# B&R Automation Studio project Laba_2
Automation Studio 4.2.5.388

## Configuration SampleText

### Task classes (Cpu.sw)
```
Cyclic#4:
  Program <- Program.prg
Libraries: sys_lib, Runtime, asstring, DriveLib
```

### Hardware
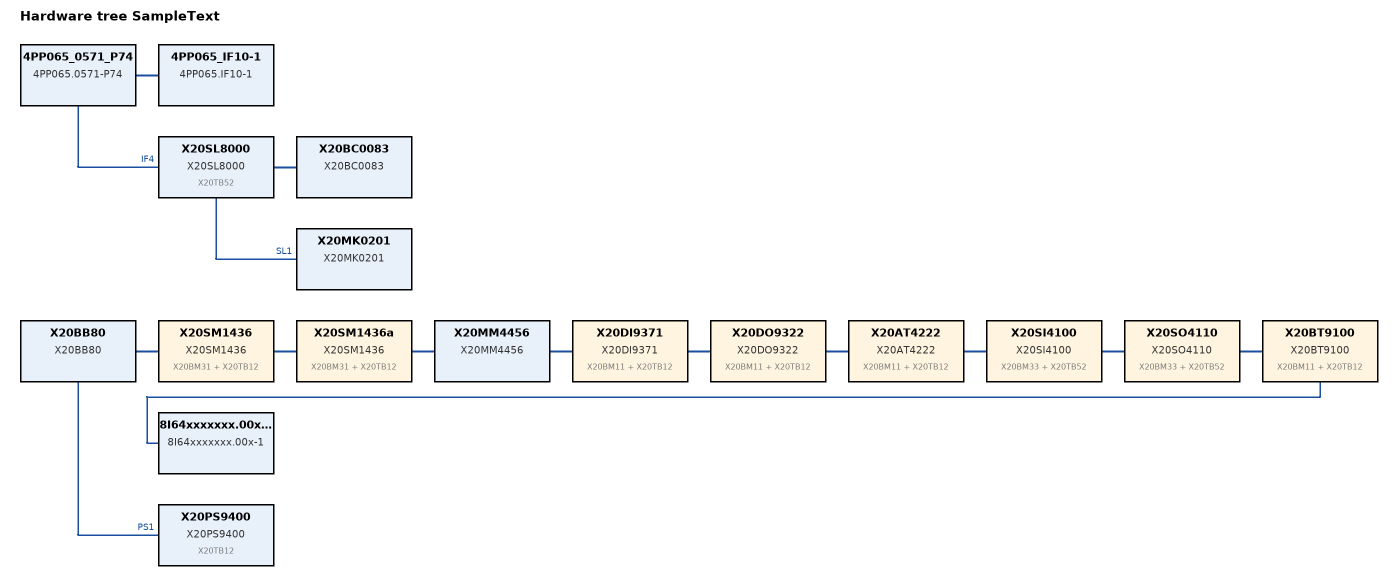
```
4PP065_0571_P74 : 4PP065.0571-P74 v1.1.2.0
  Connector IF4:
    EplInterfaceRedundant = 0
    EplEthInterfaceRedundant = 0
  Connector IF5:
    ActivateDevice = 1
    Mode = Manual
    InternetAddress = 10.0.1.10
    SubnetMask = 255.255.255.0
  ConfigurationID = labBR
  TimerDeviceType = EPLX2X
  TimerDevice = 4PP065_0571_P74.IF4
  TaskClassIdleTime = 2000
  Cyclic1Duration = 2000
  Cyclic1Tolerance = 0
  Cyclic1Output = 1
4PP065_IF10-1 : 4PP065.IF10-1 v1.0.3.0  [SS -> 4PP065_0571_P74.SS1]
8I64xxxxxxx.00x-1 : 8I64xxxxxxx.00x-1 v1.3.9.1  [X2X1 -> X20BT9100.X2X1 [Cable Type=X2XCable, Length=10, Version=1.0.0.2]]
  FunctionModel = Standard
  packedETAD = packed
  packedETI = packed
  packedCMDD = packed
  packedCMI = packed
  UNS = 220
  NCR = 10
  NSP = 890
  COS = 64
  RSC = 33000
X20AT4222 : X20AT4222 v1.2.3.0  [SS1 -> X20TB12e.SS; SL -> X20BM11c.SL1]
X20BB80 : X20BB80 v1.0.2.0
X20BC0083 : X20BC0083 v2.9.0.0  [PLK1 -> X20SL8000.PLK2 (NodeNumber=2) [Cable Type=PowerlinkCable, Length=10, Version=1.0.0.2]; SL -> X20BB80.SL1]
X20BM11 : X20BM11 v1.0.0.1  [X2X1 -> X20BM33a.X2X2]
X20BM11a : X20BM11 v1.0.0.1  [X2X1 -> X20MM4456.X2X2]
X20BM11b : X20BM11 v1.0.0.1  [X2X1 -> X20BM11a.X2X2]
X20BM11c : X20BM11 v1.0.0.1  [X2X1 -> X20BM11b.X2X2]
X20BM31 : X20BM31 v1.0.0.1  [X2X1 -> X20BB80.IF1]
X20BM31a : X20BM31 v1.0.0.1  [X2X1 -> X20BM31.X2X2]
X20BM33 : X20BM33 v1.0.0.4  [X2X1 -> X20BM11c.X2X2]
X20BM33a : X20BM33 v1.0.0.4  [X2X1 -> X20BM33.X2X2]
X20BT9100 : X20BT9100 v1.0.3.0  [SS1 -> X20TB12f.SS; SL -> X20BM11.SL1]
X20DI9371 : X20DI9371 v1.0.2.0  [SS1 -> X20TB12c.SS; SL -> X20BM11a.SL1]
X20DO9322 : X20DO9322 v1.0.3.0  [SS1 -> X20TB12d.SS; SL -> X20BM11b.SL1]
X20MK0201 : X20MK0201 v1.0.0.0  [SL -> X20SL8000.SL1]
X20MM4456 : X20MM4456 v1.1.5.0  [X2X1 -> X20BM31a.X2X2]
X20PS9400 : X20PS9400 v1.0.2.4  [SS1 -> X20TB12.SS; PS -> X20BB80.PS1]
X20SI4100 : X20SI4100 v1.10.1.1  [SS1 -> X20TB52.SS; SL -> X20BM33.SL1]
X20SL8000 : X20SL8000 v1.6.5.1  [PLK1 -> 4PP065_0571_P74.IF4 (NodeNumber=1) [Cable Type=PowerlinkCable, Length=10, Version=1.0.0.2]; PLK2 -> X20BC0083.PLK1 (NodeNumber=1) [Cable Type=PowerlinkCable, Length=10, Version=1.0.0.2]; SS1 -> X20TB52b.SS]
  SafeProject = SafeLOGIC-1
X20SM1436 : X20SM1436 v2.2.0.0  [SS1 -> X20TB12a.SS; SL -> X20BM31.SL1]
X20SM1436a : X20SM1436 v2.2.0.0  [SS1 -> X20TB12b.SS; SL -> X20BM31a.SL1]
X20SO4110 : X20SO4110 v1.10.1.1  [SS1 -> X20TB52a.SS; SL -> X20BM33a.SL1]
  SafeModuleID = 3
X20TB12 : X20TB12 v1.0.0.0
X20TB12a : X20TB12 v1.0.0.0
X20TB12b : X20TB12 v1.0.0.0
X20TB12c : X20TB12 v1.0.0.0
X20TB12d : X20TB12 v1.0.0.0
X20TB12e : X20TB12 v1.0.0.0
X20TB12f : X20TB12 v1.0.0.0
X20TB52 : X20TB52 v1.0.0.1
X20TB52a : X20TB52 v1.0.0.1
X20TB52b : X20TB52 v1.0.0.1
```

### IoMap.iom - 4PP065_0571_P74/IoMap.iom
```iecst
VAR_CONFIG
	::Program:doorSM.direction AT %IX."X20DI9371".DigitalInput01;
	::Program:StateMashine.state AT %IW."8I64xxxxxxx.00x-1".ETAD_Input;
	::Program:StateMashine.command AT %QW."8I64xxxxxxx.00x-1".CMDD_Output;
	::Program:StateMashine.speed AT %QW."8I64xxxxxxx.00x-1".LFRD_Output;
	::Program:doorSM.sw1 AT %IX."X20DI9371".DigitalInput02;
	::Program:doorSM.sw2 AT %IX."X20DI9371".DigitalInput03;
	::Program:doorSM.sw3 AT %IX."X20DI9371".DigitalInput04;
	::Program:doorSM.sw4 AT %IX."X20DI9371".DigitalInput05;
	::Program:ledSM.led1 AT %QX."X20DO9322".DigitalOutput02;
	::Program:ledSM.led2 AT %QX."X20DO9322".DigitalOutput03;
	::Program:ledSM.led3 AT %QX."X20DO9322".DigitalOutput04;
	::Program:ledSM.led4 AT %QX."X20DO9322".DigitalOutput05;
END_VAR
```

## Logical view

Binary libraries used (declarations not repeated): Runtime, Operator, AsIecCon, astime, sys_lib, asstring


### Program Logical/Program (ANSIC)

#### Variables.var
```iecst
VAR
	StateMashine : DriveStateMashine := (0);
	doorSM : DoorStateMashine := (0);
	ledSM : LedStateMashine := (0);
END_VAR
```

#### Main.c
```c
#include <bur/plctypes.h>

#ifdef _DEFAULT_INCLUDES
	#include <AsDefault.h>
#endif

void _INIT ProgramInit(void)
{
	StateMashine.enable = 1;
}

void _CYCLIC ProgramCyclic(void)
{
	DoorStateMashine(&doorSM);
	DriveStateMashine(&StateMashine);
	LedStateMashine(&ledSM);
	StateMashine.speed = doorSM.speed;
	ledSM.state = doorSM.state;
}

void _EXIT ProgramExit(void)
{

}
```

### Library Logical/DriveLib (ANSIC)

#### Types.typ
```iecst
TYPE
	States :
		(
		st_init,
		st_unknown,
		st_open,
		st_close,
		st_acc_pos,
		st_acc_neg,
		st_pos,
		st_neg,
		st_dec_pos,
		st_dec_neg
		);
END_TYPE
```

#### Constants.var
```iecst
VAR CONSTANT
	cmd_switched_on : UINT := 7;
	cmd_enabled : UINT := 15;
	cmd_shutdown : UINT := 6;
	state_disabled : UINT := 64;
	state_ready : UINT := 33;
	state_switched_on : UINT := 35;
END_VAR
```

#### DriveLib.fun
```iecst
{REDUND_ERROR} FUNCTION_BLOCK DriveStateMashine (*TODO: Add your comment here*) (*$GROUP=User,$CAT=User,$GROUPICON=User.png,$CATICON=User.png*)
	VAR_INPUT
		state : UINT;
		enable : BOOL;
	END_VAR
	VAR_OUTPUT
		command : {REDUND_UNREPLICABLE} UINT;
		speed : {REDUND_UNREPLICABLE} INT;
	END_VAR
END_FUNCTION_BLOCK

{REDUND_ERROR} FUNCTION_BLOCK DoorStateMashine (*TODO: Add your comment here*) (*$GROUP=User,$CAT=User,$GROUPICON=User.png,$CATICON=User.png*)
	VAR_INPUT
		state : UINT;
		sw1 : BOOL;
		sw2 : BOOL;
		sw3 : BOOL;
		sw4 : BOOL;
		direction : BOOL;
	END_VAR
	VAR_OUTPUT
		speed : {REDUND_UNREPLICABLE} INT;
	END_VAR
	VAR
		sw01 : BOOL;
		sw02 : BOOL;
		sw03 : BOOL;
		sw04 : BOOL;
	END_VAR
END_FUNCTION_BLOCK

{REDUND_ERROR} FUNCTION_BLOCK LedStateMashine (*TODO: Add your comment here*) (*$GROUP=User,$CAT=User,$GROUPICON=User.png,$CATICON=User.png*)
	VAR_INPUT
		state : UINT;
	END_VAR
	VAR_OUTPUT
		led1 : {REDUND_UNREPLICABLE} BOOL;
		led2 : {REDUND_UNREPLICABLE} BOOL;
		led3 : {REDUND_UNREPLICABLE} BOOL;
		led4 : {REDUND_UNREPLICABLE} BOOL;
		timer : {REDUND_UNREPLICABLE} INT;
	END_VAR
END_FUNCTION_BLOCK
```

#### DoorStateMashine.c
```c
#include <bur/plctypes.h>
#ifdef __cplusplus
	extern "C"
	{
#endif
	#include "DriveLib.h"
#ifdef __cplusplus
	};
#endif
/* TODO: Add your comment here */
void DoorStateMashine(struct DoorStateMashine* inst)
{
	/*TODO: Add your code here*/
	switch(inst->state) {
		case st_init:
			if(inst->sw1==0 && inst->sw2==0 && inst->sw3==0 && inst->sw4==0)
				inst->state = st_unknown;
			break;

		case st_unknown:
			if(inst->direction==0 && inst->sw1!=inst->sw01)
				inst->state = st_close;
			if(inst->direction==1 && inst->sw1!=inst->sw01)
				inst->state = st_neg;
			if(inst->direction==1 && inst->sw2!=inst->sw02)
				inst->state = st_acc_neg;
			if(inst->direction==1 && inst->sw3!=inst->sw03)
				inst->state = st_dec_neg;
			if(inst->direction==1 && inst->sw4!=inst->sw04)
				inst->state = st_open;
			if(inst->direction==0 && inst->sw4!=inst->sw04)
				inst->state = st_pos;
			if(inst->direction==0 && inst->sw3!=inst->sw03)
				inst->state = st_acc_pos;
			if(inst->direction==0 && inst->sw2!=inst->sw02)
				inst->state = st_dec_pos;
			break;

		case st_close:
			inst->speed = 0;
			if(inst->direction==1)
				inst->state = st_neg;
			break;

		case st_neg:
			inst->speed = -250;
			if(inst->direction==1 && inst->sw2!=inst->sw02)
				inst->state = st_acc_neg;
			if(inst->direction==0)
				inst->state = st_dec_pos;
			break;

		case st_acc_neg:
			inst->speed = -800;
			if(inst->direction==1 && inst->sw3!=inst->sw03)
				inst->state = st_dec_neg;
			if(inst->direction==0)
				inst->state = st_acc_pos;
			break;

		case st_dec_neg:
			inst->speed = -250;
			if(inst->direction==1 && inst->sw4!=inst->sw04)
				inst->state = st_open;
			if(inst->direction==0)
				inst->state = st_pos;
			break;

		case st_open:
			inst->speed = 0;
			if(inst->direction==0)
				inst->state = st_pos;
			break;

		case st_pos:
			inst->speed = 250;
			if(inst->direction==0 && inst->sw3!=inst->sw03)
				inst->state = st_acc_pos;
			if(inst->direction==1)
				inst->state = st_dec_neg;
			break;

		case st_acc_pos:
			inst->speed = 800;
			if(inst->direction==0 && inst->sw2!=inst->sw02)
				inst->state = st_dec_pos;
			if(inst->direction==1)
				inst->state = st_acc_neg;
			break;

		case st_dec_pos:
			inst->speed = 250;
			if(inst->direction==0 && inst->sw1!=inst->sw01)
				inst->state = st_close;
			if(inst->direction==1)
				inst->state = st_neg;
			break;
	}
	inst->sw01 = inst->sw1;
	inst->sw02 = inst->sw2;
	inst->sw03 = inst->sw3;
	inst->sw04 = inst->sw4;
}
```

#### DriveStateMashine.c
```c
#include <bur/plctypes.h>
#ifdef __cplusplus
	extern "C"
	{
#endif
	#include "DriveLib.h"
#ifdef __cplusplus
	};
#endif
/* TODO: Add your comment here */
void DriveStateMashine(struct DriveStateMashine* inst)
{
	/*TODO: Add your code here*/
	UINT mask = inst->state & 0x6F;
	if (inst->enable) {
		switch(mask) {
			case state_disabled:
				inst->command = cmd_shutdown;
				break;

			case state_ready:
				inst->command = cmd_enabled;
				break;

			case state_switched_on:
				inst->command = cmd_switched_on;
				break;

		}
	}
	else {
		inst->command = cmd_shutdown;
	}
}
```

#### LedStateMashine.c
```c
#include <bur/plctypes.h>
#ifdef __cplusplus
	extern "C"
	{
#endif
	#include "DriveLib.h"
#ifdef __cplusplus
	};
#endif
/* TODO: Add your comment here */
void LedStateMashine(struct LedStateMashine* inst)
{
	/*TODO: Add your code here*/
	switch(inst->state) {
		case st_init:
				break;

		case st_unknown:
			if(inst->timer % 10 == 1){
					inst->led1 = !inst->led1;
					inst->led2 = !inst->led2;
					inst->led3 = !inst->led3;
					inst->led4 = !inst->led4;
			}
			break;

		case st_close:
			inst->led1 = 1;
			inst->led2 = 1;
			inst->led3 = 1;
			inst->led4 = 1;
			break;

		case st_neg:
			inst->led1 = 0;
			if(inst->timer % 10 == 1) inst->led2 = !inst->led2;
			inst->led3 = 1;
			inst->led4 = 1;
			break;

		case st_acc_neg:
			inst->led1 = 0;
			inst->led2 = 0;
			if(inst->timer % 10 == 1) inst->led3 = !inst->led3;
			inst->led4 = 1;
			break;

		case st_dec_neg:
			inst->led1 = 0;
			inst->led2 = 0;
			inst->led3 = 0;
			if(inst->timer % 10 == 1) inst->led4 = !inst->led4;
			break;

		case st_open:
			inst->led1 = 0;
			inst->led2 = 0;
			inst->led3 = 0;
			inst->led4 = 0;
			break;

		case st_pos:
			inst->led1 = 0;
			inst->led2 = 0;
			if(inst->timer % 10 == 1) inst->led3 = !inst->led3;
			inst->led4 = 1;
			break;

		case st_acc_pos:
			inst->led1 = 0;
			if(inst->timer % 10 == 1) inst->led2 = !inst->led2;
			inst->led3 = 1;
			inst->led4 = 1;
			break;

		case st_dec_pos:
			if(inst->timer % 10 == 1) inst->led1 = !inst->led1;
			inst->led2 = 1;
			inst->led3 = 1;
			inst->led4 = 1;
			break;
	}
	inst->timer++;
}
```

Listed in the project but not available here: Logical/Global.typ, Logical/Global.var
